// TIA Portal V19 export
VAR_GLOBAL   // PLC tag table "tags_Omriktare"
   Forward AT %M0.0 : Bool;   // Command
   Backward AT %M0.1 : Bool;   // Command
   Acknowledge AT %M0.2 : Bool;   // Command
   SpeedRequest AT %MW2 : Int;   // Command
   TorqueRequest AT %MW4 : Int;   // Command
   Status AT %MW6 : Word;   // Status
   Speed_CV AT %MW8 : Int;   // Status
   Torque_CV AT %MW10 : Int;   // Status
   Alarm AT %M0.3 : Bool;   // Status
   Alarm_number AT %MW12 : Int;   // Status
END_VAR
